Fanuc KAREL source: kt00274.KL

-- PROVISIONAL review KL for V770-1; original PC SHA256 d33e75d113c4a604771d703d9146d9d5a832e38569060f7fd5690b5344ae4e81
-- Incomplete behavior may be omitted. Consult companion uncertainty JSON. Do not deploy.
PROGRAM KT00274
%NOLOCKGROUP
VAR
  OUT : BOOLEAN
-- UNRESOLVED_DECL H1 type=002017
-- UNRESOLVED_DECL H2 type=002017
BEGIN
  -- UNRESOLVED_PC offsets 5-19; opcodes 2E,22,9D,33,B4
  -- UNRESOLVED_PC offsets 24-38; opcodes 2E,22,9D,33,B4
  -- UNRESOLVED_PC offsets 43-57; opcodes 2E,22,9D,33,B4
  -- UNRESOLVED_PC offsets 62-76; opcodes 2E,22,9D,33,B4
  -- UNRESOLVED_PC offsets 81-106; opcodes 22,9D,33,B3,22,9D,33,B3,57,23
  -- UNRESOLVED_PC offsets 111-115; opcodes 7F
END KT00274
